// TIA Portal project "GR36_BP_BeltConveyorGreenx3" (V17)

(* hardware
DEVICE "ET 200SP station_1"  ET 200SP-Station
   slot 0: "Rack_0"  Rack  6ES5 710-8MAx1
   slot 1: "PLC_1"  CPU 1510SP-1 PN  6ES7 510-1DJ01-0AB0  V2.1
      slot 32768: "PROFINET interface_1"  X1
   slot 2: "DI 16x24VDC ST_1"  DI 16x24VDC ST  6ES7 131-6BH01-0BA0  V0.0
      slot 1: "DI 16x24VDC ST_1"  DI 16x24VDC ST
   slot 3: "DQ 8x24VDC/0.5A ST_1"  DQ 8x24VDC/0.5A ST  6ES7 132-6BF00-0BA0  V1.1
      slot 1: "DQ 8x24VDC/0.5A ST_1"  DQ 8x24VDC/0.5A ST
   slot 4: "AI 2xU/I 2-,4-wire HF_1"  AI 2xU/I 2-,4-wire HF  6ES7 134-6HB00-0CA1  V2.0
      slot 1: "AI 2xU/I 2-,4-wire HF_1"  AI 2xU/I 2-,4-wire HF
   slot 5: "Server module_1"  Server module  6ES7 193-6PA00-0AA0  V1.1
      slot 1: "Server module_1"  Server module
   slot 127: "BA 2xRJ45"  BA 2xRJ45  6ES7 193-6AR00-0AA0  V0.0
      slot 32769: "Port_1"  X1 P1  6ES7 193-6AR00-0AA0
      slot 32770: "Port_2"  X1 P2  6ES7 193-6AR00-0AA0
*)

// ===== PLC "PLC_1"  CPU 1510SP-1 PN =====

VAR_GLOBAL   // PLC tag table "Default tag table"
   "Clock_Byte" AT %MB69 : Byte;
   "Clock_10Hz" AT %M69.0 : Bool;
   "Clock_5Hz" AT %M69.1 : Bool;
   "Clock_2.5Hz" AT %M69.2 : Bool;
   "Clock_2Hz" AT %M69.3 : Bool;
   "Clock_1.25Hz" AT %M69.4 : Bool;
   "Clock_1Hz" AT %M69.5 : Bool;
   "Clock_0.625Hz" AT %M69.6 : Bool;
   "Clock_0.5Hz" AT %M69.7 : Bool;
   "System_Byte" AT %MB70 : Byte;
   "FirstScan" AT %M70.0 : Bool;
   "DiagStatusUpdate" AT %M70.1 : Bool;
   "AlwaysTRUE" AT %M70.2 : Bool;
   "AlwaysFALSE" AT %M70.3 : Bool;
END_VAR

VAR_GLOBAL   // PLC tag table "DigitalOutput_FactoryIO"
   "dq_Forward_M0" AT %Q0.0 : Bool;
   "dq_Backward_M0" AT %Q0.1 : Bool;
   "dq_H1" AT %Q0.2 : Bool;
   "dq_H2" AT %Q0.3 : Bool;
   "dq_H3" AT %Q0.4 : Bool;
   "dq_Horn" AT %Q0.5 : Bool;
   "dq_Forward_M1" AT %Q1.0 : Bool;
   "dq_Forward_M2" AT %Q1.4 : Bool;
END_VAR

VAR_GLOBAL   // PLC tag table "DigitalInput_FactoryIO"
   "di_AtLeft" AT %I0.0 : Bool;
   "di_AtMiddle" AT %I0.1 : Bool;
   "di_AtRight" AT %I0.2 : Bool;
   "di_IsHight" AT %I0.3 : Bool;
   "di_SwtichBay3" AT %I0.6 : Bool;
   "di_Measure" AT %I0.4 : Bool;
   "di_ImpulsFromShaft" AT %I0.5 : Bool;
   "di_FactoryIO_Running" AT %I0.7 : Bool;
   "di_AtExit_B11" AT %I1.0 : Bool;
   "di_AtExit_B22" AT %I1.4 : Bool;
END_VAR

VAR_GLOBAL   // PLC tag table "DigitalOutput_PLC"
   "dq_LedWhite" AT %Q4.2 : Bool;
   "dq_LedBlue" AT %Q4.3 : Bool;
   "dq_LedGreen" AT %Q4.0 : Bool;
   "dq_LedRed" AT %Q4.1 : Bool;
END_VAR

VAR_GLOBAL   // PLC tag table "DigitalInput_PLC"
   "di_StartButton" AT %I51.0 : Bool;
   "di_StopButton" AT %I51.1 : Bool;
   "di_Selector" AT %I51.2 : Bool;
   "di_ResetButton" AT %I51.3 : Bool;
   "di_Switch_M0" AT %I50.0 : Bool;
   "di_Switch_M1" AT %I50.1 : Bool;
   "di_Switch_M2" AT %I50.2 : Bool;
END_VAR

VAR_GLOBAL   // PLC tag table "ErrorCodes"
   "mw_ErrorCode" AT %MW100 : Word;
   "m_ErrorConveyor_M0" AT %M101.0 : Bool;
   "m_ErrorConveyor_M1" AT %M101.1 : Bool;
   "m_ErrorConveyor_M2" AT %M101.2 : Bool;
END_VAR

TYPE "edge_detection"
   STRUCT
      memory : Struct
         LastState_Positive : Bool;
         LastState_Negative : Bool;
      END_STRUCT;
      OneShoot_Positive : Bool;
      OneShoot_Negative : Bool;
   END_STRUCT;
END_TYPE

DATA_BLOCK "db_Mode"   // DB1
{ S7_Optimized_Access := 'TRUE' }
VERSION : 0.1
   VAR
      Auto : Bool;
      Manual : Bool;
      GlobalError : Bool;
   END_VAR
BEGIN
END_DATA_BLOCK

DATA_BLOCK "db_Output"   // DB2
{ S7_Optimized_Access := 'TRUE' }
VERSION : 0.1
   VAR
      M0_Forward_Auto : Bool;
      M1_Forward_Auto : Bool;
      M2_Forward_Auto : Bool;
      M0_Forward_Manual : Bool;
      M1_Forward_Manual : Bool;
      M2_Forward_Manual : Bool;
   END_VAR
BEGIN
END_DATA_BLOCK

DATA_BLOCK "db_Conveyor"   // DB3
{ S7_Optimized_Access := 'TRUE' }
VERSION : 0.1
   VAR
      isM1Occupied : Bool;
      isM2Occupied : Bool;
   END_VAR
BEGIN
END_DATA_BLOCK

DATA_BLOCK "db_Edge"   // DB4
{ S7_Optimized_Access := 'TRUE' }
VERSION : 0.1
   VAR
      AtRight : "edge_detection";
      AtExit_B11 : "edge_detection";
      AtExit_B22 : "edge_detection";
   END_VAR
BEGIN
END_DATA_BLOCK

DATA_BLOCK "db_Settings"   // DB7
{ S7_Optimized_Access := 'TRUE' }
VERSION : 0.1
   VAR
      ErrorCodeDelay : Time := t#3s;
      M0Delay : Time := T#15s;
      M1Delay : Time := t#8s;
      M2Delay : Time := t#8s;
   END_VAR
BEGIN
END_DATA_BLOCK

// folder: System blocks/Program resources

DATA_BLOCK "c_signalizationBlueLightErrorcode"   // DB5
{ S7_Optimized_Access := 'TRUE' }
AUTHOR : Simatic
FAMILY : IEC
NAME : CNTR
VERSION : 1.0
// stored: InstanceOfName IEC_COUNTER
"IEC_COUNTER"
BEGIN
END_DATA_BLOCK

DATA_BLOCK "t_count3sDelayInErrorCode"   // DB6
{ S7_Optimized_Access := 'TRUE' }
AUTHOR : Simatic
FAMILY : IEC
NAME : IEC_TMR
VERSION : 1.0
// stored: InstanceOfName IEC_TIMER
"IEC_TIMER"
BEGIN
END_DATA_BLOCK

DATA_BLOCK "t_M0_travelsal"   // DB8
{ S7_Optimized_Access := 'TRUE' }
AUTHOR : Simatic
FAMILY : IEC
NAME : IEC_TMR
VERSION : 1.0
// stored: InstanceOfName IEC_TIMER
"IEC_TIMER"
BEGIN
END_DATA_BLOCK

DATA_BLOCK "t_M2_Traversal"   // DB9
{ S7_Optimized_Access := 'TRUE' }
AUTHOR : Simatic
FAMILY : IEC
NAME : IEC_TMR
VERSION : 1.0
// stored: InstanceOfName IEC_TIMER
"IEC_TIMER"
BEGIN
END_DATA_BLOCK

DATA_BLOCK "t_M1_travelsal"   // DB10
{ S7_Optimized_Access := 'TRUE' }
AUTHOR : Simatic
FAMILY : IEC
NAME : IEC_TMR
VERSION : 1.0
// stored: InstanceOfName IEC_TIMER
"IEC_TIMER"
BEGIN
END_DATA_BLOCK

// folder: (top level)

FUNCTION "fc_Mode" : Void   // FC1, LAD
{ S7_Optimized_Access := 'TRUE' }
VERSION : 0.1
BEGIN

REGION Network 1: Auto
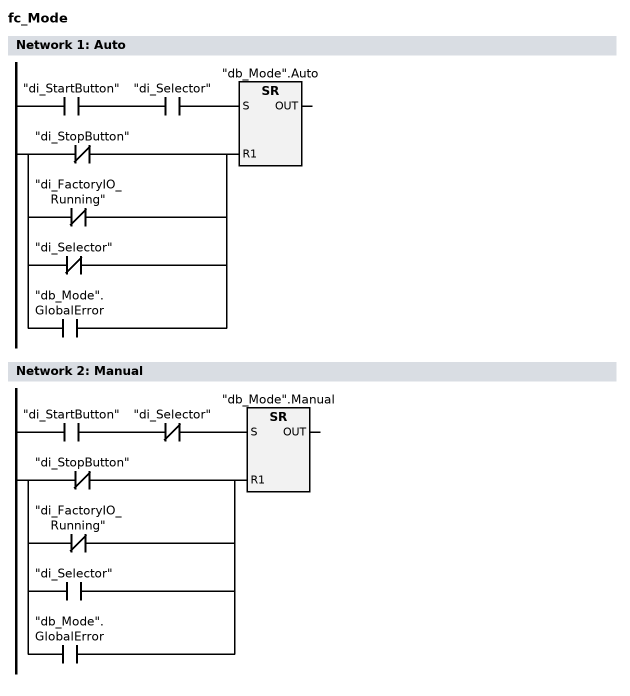
   RUNG wire#powerrail
      Contact( "di_StartButton" )
      Contact( "di_Selector" )
      S_SR(operand := "db_Mode".Auto, r1 := wire#w1)
   END_RUNG
   RUNG wire#powerrail
      I_Contact( "di_StopButton" )
   END_RUNG wire#w1
   RUNG wire#powerrail
      I_Contact( "di_FactoryIO_Running" )
   END_RUNG wire#w1
   RUNG wire#powerrail
      I_Contact( "di_Selector" )
   END_RUNG wire#w1
   RUNG wire#powerrail
      Contact( "db_Mode".GlobalError )
   END_RUNG wire#w1
   // the same network as SCL:
   IF "di_StartButton" AND "di_Selector" THEN
       "db_Mode".Auto := TRUE;   // SR flip-flop
   END_IF;
   IF NOT "di_StopButton" OR NOT "di_FactoryIO_Running" OR NOT "di_Selector" OR "db_Mode".GlobalError THEN
       "db_Mode".Auto := FALSE;
   END_IF;
END_REGION

REGION Network 2: Manual
   RUNG wire#powerrail
      Contact( "di_StartButton" )
      I_Contact( "di_Selector" )
      S_SR(operand := "db_Mode".Manual, r1 := wire#w1)
   END_RUNG
   RUNG wire#powerrail
      I_Contact( "di_StopButton" )
   END_RUNG wire#w1
   RUNG wire#powerrail
      I_Contact( "di_FactoryIO_Running" )
   END_RUNG wire#w1
   RUNG wire#powerrail
      Contact( "di_Selector" )
   END_RUNG wire#w1
   RUNG wire#powerrail
      Contact( "db_Mode".GlobalError )
   END_RUNG wire#w1
   // the same network as SCL:
   IF "di_StartButton" AND NOT "di_Selector" THEN
       "db_Mode".Manual := TRUE;   // SR flip-flop
   END_IF;
   IF NOT "di_StopButton" OR NOT "di_FactoryIO_Running" OR "di_Selector" OR "db_Mode".GlobalError THEN
       "db_Mode".Manual := FALSE;
   END_IF;
END_REGION
END_FUNCTION

FUNCTION "fc_Output" : Void   // FC2, LAD
{ S7_Optimized_Access := 'TRUE' }
VERSION : 0.1
BEGIN

REGION Network 1: M0
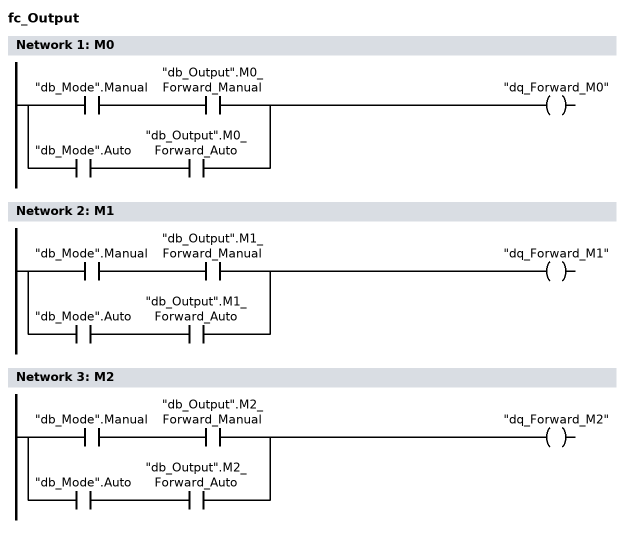
   RUNG wire#powerrail
      Contact( "db_Mode".Manual )
      Contact( "db_Output".M0_Forward_Manual )
      wire#w1
      Coil( "dq_Forward_M0" )
   END_RUNG
   RUNG wire#powerrail
      Contact( "db_Mode".Auto )
      Contact( "db_Output".M0_Forward_Auto )
   END_RUNG wire#w1
   // the same network as SCL:
   "dq_Forward_M0" := ("db_Mode".Manual AND "db_Output".M0_Forward_Manual) OR ("db_Mode".Auto AND "db_Output".M0_Forward_Auto);
END_REGION

REGION Network 2: M1
   RUNG wire#powerrail
      Contact( "db_Mode".Manual )
      Contact( "db_Output".M1_Forward_Manual )
      wire#w1
      Coil( "dq_Forward_M1" )
   END_RUNG
   RUNG wire#powerrail
      Contact( "db_Mode".Auto )
      Contact( "db_Output".M1_Forward_Auto )
   END_RUNG wire#w1
   // the same network as SCL:
   "dq_Forward_M1" := ("db_Mode".Manual AND "db_Output".M1_Forward_Manual) OR ("db_Mode".Auto AND "db_Output".M1_Forward_Auto);
END_REGION

REGION Network 3: M2
   RUNG wire#powerrail
      Contact( "db_Mode".Manual )
      Contact( "db_Output".M2_Forward_Manual )
      wire#w1
      Coil( "dq_Forward_M2" )
   END_RUNG
   RUNG wire#powerrail
      Contact( "db_Mode".Auto )
      Contact( "db_Output".M2_Forward_Auto )
   END_RUNG wire#w1
   // the same network as SCL:
   "dq_Forward_M2" := ("db_Mode".Manual AND "db_Output".M2_Forward_Manual) OR ("db_Mode".Auto AND "db_Output".M2_Forward_Auto);
END_REGION
END_FUNCTION

FUNCTION "fc_Manual" : Void   // FC3, LAD
{ S7_Optimized_Access := 'TRUE' }
VERSION : 0.1
BEGIN

REGION Network 1: M0
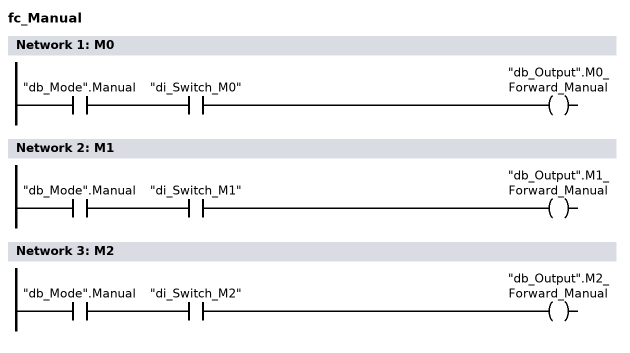
   RUNG wire#powerrail
      Contact( "db_Mode".Manual )
      Contact( "di_Switch_M0" )
      Coil( "db_Output".M0_Forward_Manual )
   END_RUNG
   // the same network as SCL:
   "db_Output".M0_Forward_Manual := "db_Mode".Manual AND "di_Switch_M0";
END_REGION

REGION Network 2: M1
   RUNG wire#powerrail
      Contact( "db_Mode".Manual )
      Contact( "di_Switch_M1" )
      Coil( "db_Output".M1_Forward_Manual )
   END_RUNG
   // the same network as SCL:
   "db_Output".M1_Forward_Manual := "db_Mode".Manual AND "di_Switch_M1";
END_REGION

REGION Network 3: M2
   RUNG wire#powerrail
      Contact( "db_Mode".Manual )
      Contact( "di_Switch_M2" )
      Coil( "db_Output".M2_Forward_Manual )
   END_RUNG
   // the same network as SCL:
   "db_Output".M2_Forward_Manual := "db_Mode".Manual AND "di_Switch_M2";
END_REGION
END_FUNCTION

FUNCTION "fc_LightSignalization" : Void   // FC4, LAD
{ S7_Optimized_Access := 'TRUE' }
VERSION : 0.1
BEGIN

REGION Network 1: Auto & Manual mode signalization
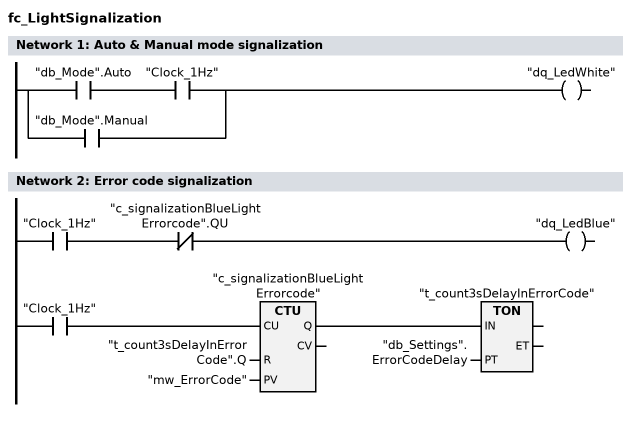
   RUNG wire#powerrail
      Contact( "db_Mode".Auto )
      Contact( "Clock_1Hz" )
      wire#w1
      Coil( "dq_LedWhite" )
   END_RUNG
   RUNG wire#powerrail
      Contact( "db_Mode".Manual )
   END_RUNG wire#w1
   // the same network as SCL:
   "dq_LedWhite" := ("db_Mode".Auto AND "Clock_1Hz") OR "db_Mode".Manual;
END_REGION

REGION Network 2: Error code signalization
   "dq_LedBlue" := "Clock_1Hz" AND NOT "c_signalizationBlueLightErrorcode".QU;
   "c_signalizationBlueLightErrorcode".CTU(CU := "Clock_1Hz",
                           R := "t_count3sDelayInErrorCode".Q,
                           PV := "mw_ErrorCode");
   "t_count3sDelayInErrorCode".TON(IN := "c_signalizationBlueLightErrorcode".Q,
                           PT := "db_Settings".ErrorCodeDelay);
END_REGION
END_FUNCTION

FUNCTION "fc_Auto" : Void   // FC5, LAD
{ S7_Optimized_Access := 'TRUE' }
VERSION : 0.1
BEGIN

REGION Network 1: M0
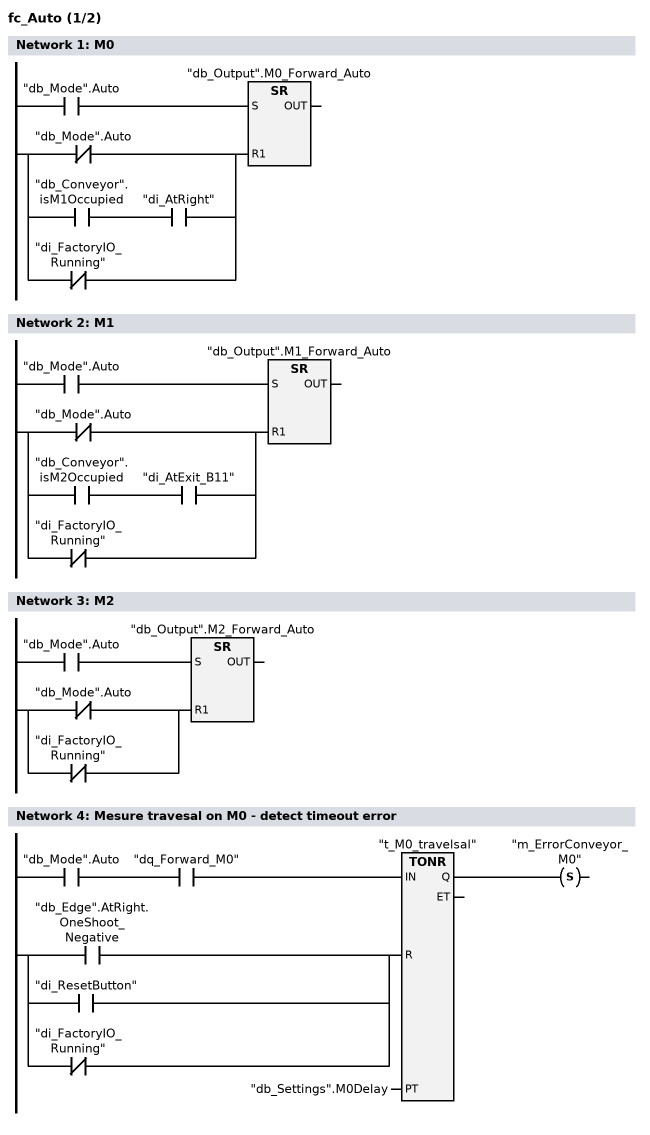
   RUNG wire#powerrail
      Contact( "db_Mode".Auto )
      S_SR(operand := "db_Output".M0_Forward_Auto, r1 := wire#w1)
   END_RUNG
   RUNG wire#powerrail
      I_Contact( "db_Mode".Auto )
   END_RUNG wire#w1
   RUNG wire#powerrail
      Contact( "db_Conveyor".isM1Occupied )
      Contact( "di_AtRight" )
   END_RUNG wire#w1
   RUNG wire#powerrail
      I_Contact( "di_FactoryIO_Running" )
   END_RUNG wire#w1
   // the same network as SCL:
   IF "db_Mode".Auto THEN
       "db_Output".M0_Forward_Auto := TRUE;   // SR flip-flop
   END_IF;
   IF NOT "db_Mode".Auto OR ("db_Conveyor".isM1Occupied AND "di_AtRight") OR NOT "di_FactoryIO_Running" THEN
       "db_Output".M0_Forward_Auto := FALSE;
   END_IF;
END_REGION

REGION Network 2: M1
   RUNG wire#powerrail
      Contact( "db_Mode".Auto )
      S_SR(operand := "db_Output".M1_Forward_Auto, r1 := wire#w1)
   END_RUNG
   RUNG wire#powerrail
      I_Contact( "db_Mode".Auto )
   END_RUNG wire#w1
   RUNG wire#powerrail
      Contact( "db_Conveyor".isM2Occupied )
      Contact( "di_AtExit_B11" )
   END_RUNG wire#w1
   RUNG wire#powerrail
      I_Contact( "di_FactoryIO_Running" )
   END_RUNG wire#w1
   // the same network as SCL:
   IF "db_Mode".Auto THEN
       "db_Output".M1_Forward_Auto := TRUE;   // SR flip-flop
   END_IF;
   IF NOT "db_Mode".Auto OR ("db_Conveyor".isM2Occupied AND "di_AtExit_B11") OR NOT "di_FactoryIO_Running" THEN
       "db_Output".M1_Forward_Auto := FALSE;
   END_IF;
END_REGION

REGION Network 3: M2
   RUNG wire#powerrail
      Contact( "db_Mode".Auto )
      S_SR(operand := "db_Output".M2_Forward_Auto, r1 := wire#w1)
   END_RUNG
   RUNG wire#powerrail
      I_Contact( "db_Mode".Auto )
   END_RUNG wire#w1
   RUNG wire#powerrail
      I_Contact( "di_FactoryIO_Running" )
   END_RUNG wire#w1
   // the same network as SCL:
   IF "db_Mode".Auto THEN
       "db_Output".M2_Forward_Auto := TRUE;   // SR flip-flop
   END_IF;
   IF NOT "db_Mode".Auto OR NOT "di_FactoryIO_Running" THEN "db_Output".M2_Forward_Auto := FALSE; END_IF;
END_REGION

REGION Network 4: Mesure travesal on M0 - detect timeout error
   "t_M0_travelsal".TONR(IN := "db_Mode".Auto AND "dq_Forward_M0",
                         R := "db_Edge".AtRight.OneShoot_Negative OR "di_ResetButton" OR NOT "di_FactoryIO_Running",
                         PT := "db_Settings".M0Delay);
   IF "t_M0_travelsal".Q THEN "m_ErrorConveyor_M0" := TRUE; END_IF;
END_REGION

REGION Network 5: Mesure travesal on M1- detect timeout error
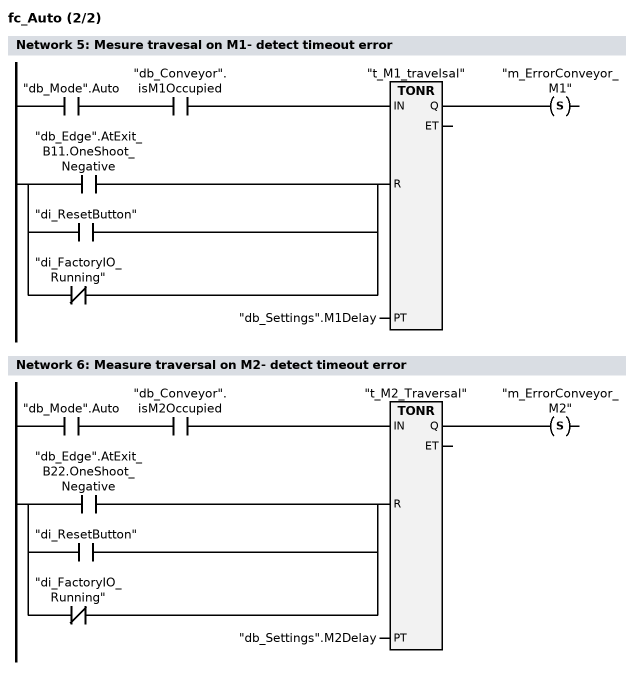
   "t_M1_travelsal".TONR(IN := "db_Mode".Auto AND "db_Conveyor".isM1Occupied,
                         R := "db_Edge".AtExit_B11.OneShoot_Negative OR "di_ResetButton" OR NOT "di_FactoryIO_Running",
                         PT := "db_Settings".M1Delay);
   IF "t_M1_travelsal".Q THEN "m_ErrorConveyor_M1" := TRUE; END_IF;
END_REGION

REGION Network 6: Measure traversal on M2- detect timeout error
   "t_M2_Traversal".TONR(IN := "db_Mode".Auto AND "db_Conveyor".isM2Occupied,
                         R := "db_Edge".AtExit_B22.OneShoot_Negative OR "di_ResetButton" OR NOT "di_FactoryIO_Running",
                         PT := "db_Settings".M2Delay);
   IF "t_M2_Traversal".Q THEN "m_ErrorConveyor_M2" := TRUE; END_IF;
END_REGION
END_FUNCTION

FUNCTION "fc_Conveyor" : Void   // FC6, LAD
{ S7_Optimized_Access := 'TRUE' }
VERSION : 0.1
BEGIN

REGION Network 1: Check if M1 is occupied
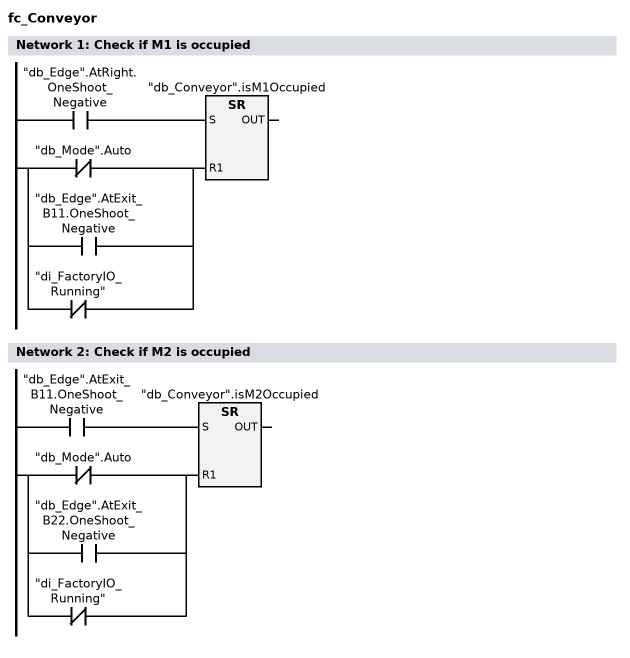
   RUNG wire#powerrail
      Contact( "db_Edge".AtRight.OneShoot_Negative )
      S_SR(operand := "db_Conveyor".isM1Occupied, r1 := wire#w1)
   END_RUNG
   RUNG wire#powerrail
      I_Contact( "db_Mode".Auto )
   END_RUNG wire#w1
   RUNG wire#powerrail
      Contact( "db_Edge".AtExit_B11.OneShoot_Negative )
   END_RUNG wire#w1
   RUNG wire#powerrail
      I_Contact( "di_FactoryIO_Running" )
   END_RUNG wire#w1
   // the same network as SCL:
   IF "db_Edge".AtRight.OneShoot_Negative THEN
       "db_Conveyor".isM1Occupied := TRUE;   // SR flip-flop
   END_IF;
   IF NOT "db_Mode".Auto OR "db_Edge".AtExit_B11.OneShoot_Negative OR NOT "di_FactoryIO_Running" THEN
       "db_Conveyor".isM1Occupied := FALSE;
   END_IF;
END_REGION

REGION Network 2: Check if M2 is occupied
   RUNG wire#powerrail
      Contact( "db_Edge".AtExit_B11.OneShoot_Negative )
      S_SR(operand := "db_Conveyor".isM2Occupied, r1 := wire#w1)
   END_RUNG
   RUNG wire#powerrail
      I_Contact( "db_Mode".Auto )
   END_RUNG wire#w1
   RUNG wire#powerrail
      Contact( "db_Edge".AtExit_B22.OneShoot_Negative )
   END_RUNG wire#w1
   RUNG wire#powerrail
      I_Contact( "di_FactoryIO_Running" )
   END_RUNG wire#w1
   // the same network as SCL:
   IF "db_Edge".AtExit_B11.OneShoot_Negative THEN
       "db_Conveyor".isM2Occupied := TRUE;   // SR flip-flop
   END_IF;
   IF NOT "db_Mode".Auto OR "db_Edge".AtExit_B22.OneShoot_Negative OR NOT "di_FactoryIO_Running" THEN
       "db_Conveyor".isM2Occupied := FALSE;
   END_IF;
END_REGION
END_FUNCTION

FUNCTION "fc_Edge" : Void   // FC7, LAD
{ S7_Optimized_Access := 'TRUE' }
VERSION : 0.1
   VAR_TEMP   // added for the SCL form of the ladder/FBD networks
      _w1 : Bool;
   END_VAR
BEGIN

REGION Network 1: AtRight
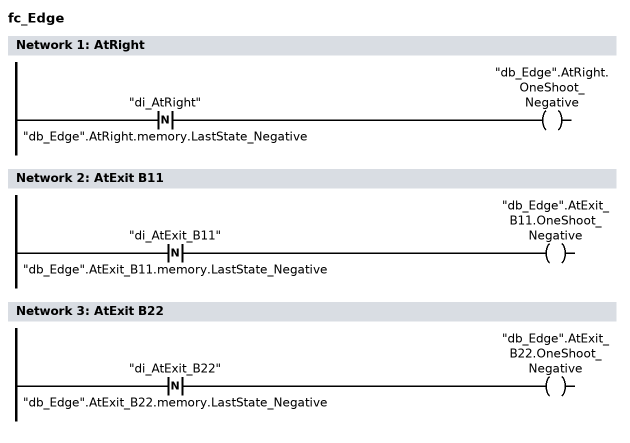
   RUNG wire#powerrail
      N_Contact(operand := "di_AtRight", bit := "db_Edge".AtRight.memory.LastState_Negative)
      Coil( "db_Edge".AtRight.OneShoot_Negative )
   END_RUNG
   // the same network as SCL:
   #_w1 := NOT "di_AtRight" AND "db_Edge".AtRight.memory.LastState_Negative;   // falling edge of "di_AtRight"
   "db_Edge".AtRight.memory.LastState_Negative := "di_AtRight";
   "db_Edge".AtRight.OneShoot_Negative := #_w1;
END_REGION

REGION Network 2: AtExit B11
   RUNG wire#powerrail
      N_Contact(operand := "di_AtExit_B11", bit := "db_Edge".AtExit_B11.memory.LastState_Negative)
      Coil( "db_Edge".AtExit_B11.OneShoot_Negative )
   END_RUNG
   // the same network as SCL:
   #_w1 := NOT "di_AtExit_B11" AND "db_Edge".AtExit_B11.memory.LastState_Negative;   // falling edge of "di_AtExit_B11"
   "db_Edge".AtExit_B11.memory.LastState_Negative := "di_AtExit_B11";
   "db_Edge".AtExit_B11.OneShoot_Negative := #_w1;
END_REGION

REGION Network 3: AtExit B22
   RUNG wire#powerrail
      N_Contact(operand := "di_AtExit_B22", bit := "db_Edge".AtExit_B22.memory.LastState_Negative)
      Coil( "db_Edge".AtExit_B22.OneShoot_Negative )
   END_RUNG
   // the same network as SCL:
   #_w1 := NOT "di_AtExit_B22" AND "db_Edge".AtExit_B22.memory.LastState_Negative;   // falling edge of "di_AtExit_B22"
   "db_Edge".AtExit_B22.memory.LastState_Negative := "di_AtExit_B22";
   "db_Edge".AtExit_B22.OneShoot_Negative := #_w1;
END_REGION
END_FUNCTION

FUNCTION "fc_Error" : Void   // FC8, LAD
{ S7_Optimized_Access := 'TRUE' }
VERSION : 0.1
BEGIN

REGION Network 1: Set global error when minor error occurs
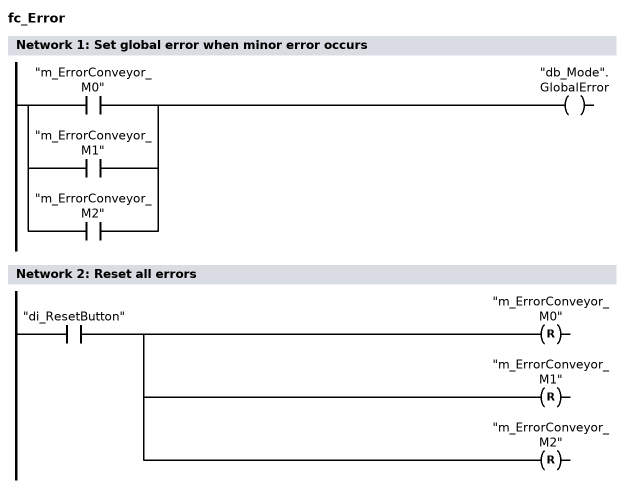
   RUNG wire#powerrail
      Contact( "m_ErrorConveyor_M0" )
      wire#w1
      Coil( "db_Mode".GlobalError )
   END_RUNG
   RUNG wire#powerrail
      Contact( "m_ErrorConveyor_M1" )
   END_RUNG wire#w1
   RUNG wire#powerrail
      Contact( "m_ErrorConveyor_M2" )
   END_RUNG wire#w1
   // the same network as SCL:
   "db_Mode".GlobalError := "m_ErrorConveyor_M0" OR "m_ErrorConveyor_M1" OR "m_ErrorConveyor_M2";
END_REGION

REGION Network 2: Reset all errors
   RUNG wire#powerrail
      Contact( "di_ResetButton" )
      wire#w1
      R_Coil( "m_ErrorConveyor_M0" )
   END_RUNG
   RUNG wire#w1
      R_Coil( "m_ErrorConveyor_M1" )
   END_RUNG
   RUNG wire#w1
      R_Coil( "m_ErrorConveyor_M2" )
   END_RUNG
   // the same network as SCL:
   IF "di_ResetButton" THEN
       "m_ErrorConveyor_M0" := FALSE;
       "m_ErrorConveyor_M1" := FALSE;
       "m_ErrorConveyor_M2" := FALSE;
   END_IF;
END_REGION
END_FUNCTION

ORGANIZATION_BLOCK "Main"   // OB1, LAD, ProgramCycle
TITLE = "Main Program Sweep (Cycle)"
{ S7_Optimized_Access := 'TRUE' }
VERSION : 0.1
   VAR_INPUT
      Initial_Call : Bool;   // Initial call of this OB
      Remanence : Bool;   // =True, if remanent data are available
   END_VAR
BEGIN

REGION Network 1
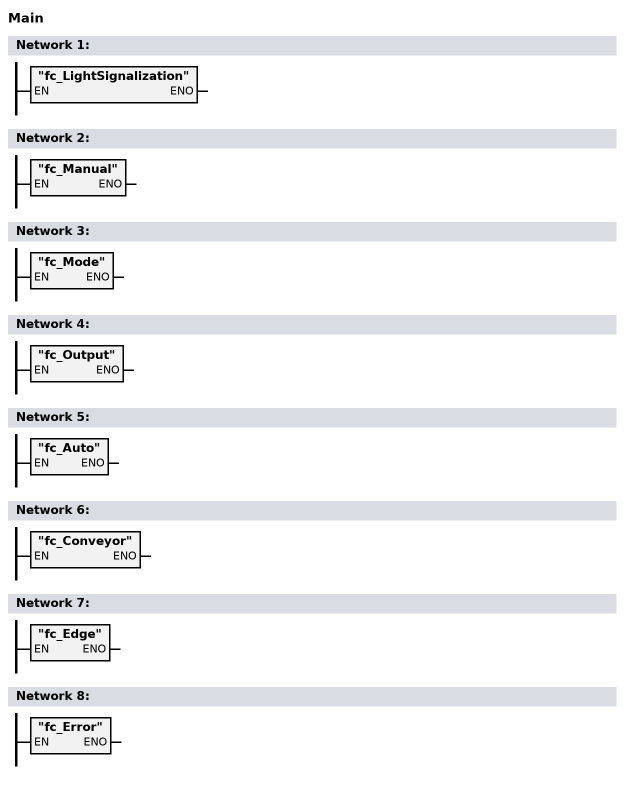
   RUNG wire#powerrail
      "fc_LightSignalization"()
   END_RUNG
   // the same network as SCL:
   "fc_LightSignalization"();
END_REGION

REGION Network 2
   RUNG wire#powerrail
      "fc_Manual"()
   END_RUNG
   // the same network as SCL:
   "fc_Manual"();
END_REGION

REGION Network 3
   RUNG wire#powerrail
      "fc_Mode"()
   END_RUNG
   // the same network as SCL:
   "fc_Mode"();
END_REGION

REGION Network 4
   RUNG wire#powerrail
      "fc_Output"()
   END_RUNG
   // the same network as SCL:
   "fc_Output"();
END_REGION

REGION Network 5
   RUNG wire#powerrail
      "fc_Auto"()
   END_RUNG
   // the same network as SCL:
   "fc_Auto"();
END_REGION

REGION Network 6
   RUNG wire#powerrail
      "fc_Conveyor"()
   END_RUNG
   // the same network as SCL:
   "fc_Conveyor"();
END_REGION

REGION Network 7
   RUNG wire#powerrail
      "fc_Edge"()
   END_RUNG
   // the same network as SCL:
   "fc_Edge"();
END_REGION

REGION Network 8
   RUNG wire#powerrail
      "fc_Error"()
   END_RUNG
   // the same network as SCL:
   "fc_Error"();
END_REGION
END_ORGANIZATION_BLOCK